Universal Robots URScript: dus_probe_l.script

# =============================================================================
#  dus_probe_l.script — dusan_v1
#  Y+ 로 너비/2 이동해 측정한다. 이 점이 원점이 된다
#
#  펜던트에서 "4_probe_left" 자리에 스크립트 노드를 파일(File) 모드로 넣고 지정한다.
#
#  ※ def main() 으로 감싸지 말 것 (펜던트가 호출하지 않는다)
#  ※ 최상위에 global 을 쓰지 말 것 (preamble 이 이미 선언·대입해 뒀다)
#  ※ if / while 은 반드시 end 로 닫을 것
# =============================================================================

# 중앙에서 Y+ 로 너비의 절반만큼
    tgt_pose = get_actual_tcp_pose()
    tgt_pose[1] = y_c + app_width * 0.0005
    movel(tgt_pose, a = 1.2, v = v_move)
    y_l = get_actual_tcp_pose()[1]

# Y+ 끝 접근
def pl_move():
  movel(tgt_pose, a = 1.2, v = v_seek)
end

x_start = get_actual_tcp_pose()[0]
tgt_pose = get_actual_tcp_pose()
tgt_pose[0] = x_start + seek_limit * 0.001
mv_h = start_thread(pl_move, (), detach_mode = False)
while (True):
  if (get_standard_digital_in(sensor_di1) and get_standard_digital_in(sensor_di2)):
    stop_thread(mv_h)
    stopl(1.2)
    break
  end
  if (get_actual_tcp_pose()[0] >= tgt_pose[0] - 0.0005):
    stop_thread(mv_h)
    stopl(1.2)
    break
  end
  sync()
end

# 센서로 멈췄는지 한계로 멈췄는지 기록 (센서가 아직 없어도 계속 진행한다)
if (get_standard_digital_in(sensor_di1) and get_standard_digital_in(sensor_di2)):
  n_hit = n_hit + 1
end
n_probe = n_probe + 1
write_port_register(304, n_probe)
write_port_register(305, n_hit)

    p_lx = get_actual_tcp_pose()[0]
    write_port_register(301, floor(p_lx * 10000 + 0.5))

    # 이 자리가 원점이다
    zero_pose = get_actual_tcp_pose()
    zero_inv = pose_inv(zero_pose)
    zero_ok = True

tgt_pose = get_actual_tcp_pose()
tgt_pose[0] = x_start
movel(tgt_pose, a = 1.2, v = v_move)
